(* PLC project controller, Dassault Systèmes ControlBuild 2024x *)
(* stored: creationDateTime 2023-10-03T11:13:48-01:00 *)

PROGRAM tni_clock.controller
  VAR_INPUT
    pressure : INT := 0;
  END_VAR
  VAR_INPUT
    tick : BOOL := false;
  END_VAR
  VAR_IN_OUT
    B1 : BOOL := false;
    B2 : BOOL := false;
    B3 : BOOL := false;
    B4 : BOOL := false;
  END_VAR
  VAR_OUTPUT
    displayValue : ARRAY[1..8] OF BYTE := [8(0)];
  END_VAR
  VAR_OUTPUT
    stepMotorSecond : BOOL := false;
    stepMotorMinute : BOOL := false;
    stepMotorHour : BOOL := false;
  END_VAR
  VAR_OUTPUT
    switchOnLight : BOOL := false;
  END_VAR

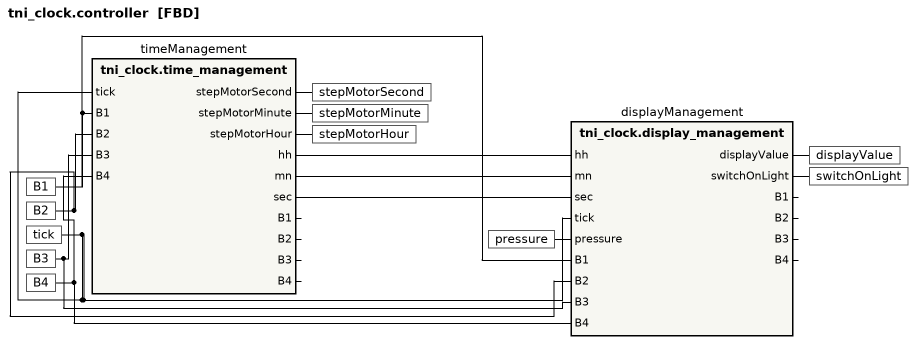
(* FBD diagram, written out as Structured Text *)
timeManagement(tick := tick, B1 := B1, B2 := B2, B3 := B3, B4 := B4);
stepMotorSecond := timeManagement.stepMotorSecond;
stepMotorMinute := timeManagement.stepMotorMinute;
stepMotorHour := timeManagement.stepMotorHour;
displayManagement(hh := timeManagement.hh, mn := timeManagement.mn, sec := timeManagement.sec, tick := tick, pressure := pressure, B1 := B1, B2 := B2, B3 := B3, B4 := B4);
displayValue := displayManagement.displayValue;
switchOnLight := displayManagement.switchOnLight;
END_PROGRAM
